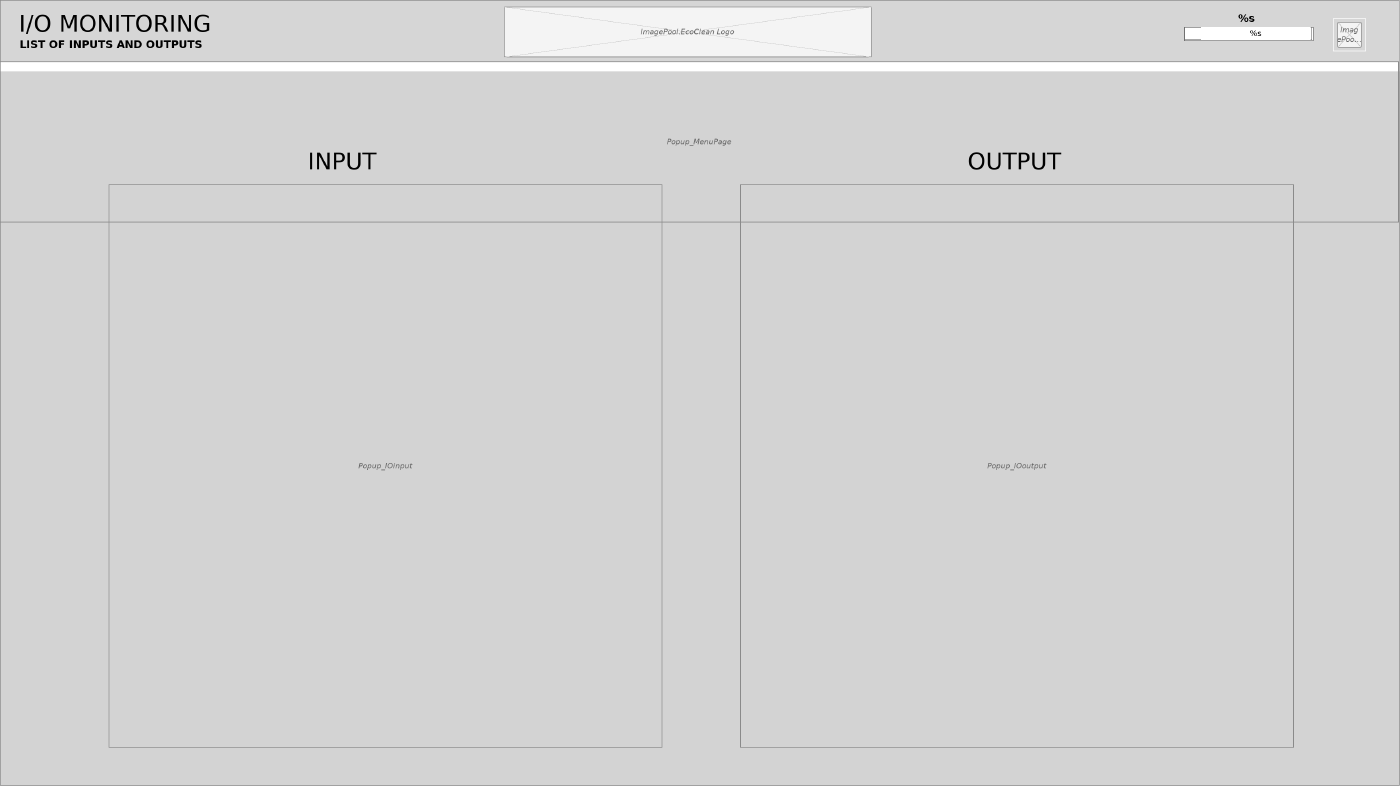
VISUALIZATION IO_Monitoring  // 1920x1079
    Rectangle (0,98 1920x981)
    Group (141,247 1639x790)
        Rectangle (0,0 774x790)
        Rectangle (865,0 774x790)
    Rectangle (0,63 1920x26)
        p3528305787: HMI_Ctrl.ANIMATION3
    Rectangle (0,0 1919x85)
    Label (23,6 310x53), "I/O MONITORING"
    Label (24,49 320x24), "LIST OF INPUTS AND OUTPUTS"
    Group (1828,25 45x45)
        OnMouseClick: toggle HMI_Ctrl.MenuButton
        RoundedRectangle (0,0 45x45), colour toggle: HMI_Ctrl.MenuButton
        Image (6,5 33x35), image: ImagePool.Menu Button
    Frame (149,253 759x773)
        shows Popup_IOinput()
    Frame (1015,253 759x773)
        shows Popup_IOoutput()
    Image (691,9 504x69), image: ImagePool.EcoClean Logo
    Group (1621,14 180x42)
        Rectangle (0,0 177x22), "%s", text variable: DSLocalSystemTimeML.sCurrentDT24Hr_General
        Button (3,23 177x19), image: VisuSymbols.Symbols.AddUser
        Rectangle (26,23 150x18), "%s", text variable: fbHmiTF1800_UserlevelManagement.dsHmiUserStatus_Active.sLoginName
    Label (419,195 125x53), "INPUT"
    Label (1324,195 153x53), "OUTPUT"
    Frame (0,84 1918x221), invisible if: HMI_Ctrl.CloseMenuButton
        shows Popup_MenuPage()
END_VISUALIZATION

(* stored: Version 1.1.0.1, ProductVersion 3.1.4024.12
   Visu IO_Monitoring: Id {fbd58c1d-0ac4-4869-8fd5-124abf61bae0} *)
